Staubli VAL3: OnF5.pgx

program OnF5()
begin
  //
  call IO:Main(0)
  bUserRefresh=true
end
